// TwinCAT 3 PLC project MachineA
// ProgramVersion: 3.1.4026.22
// CompilerDefines: VISU_USEPROPERTYINFO
// libraries:
//   [DeviceLibrary], * (MechDS)
//   Tc2_MC2, * (Beckhoff Automation GmbH)
//   Tc2_Standard, * (Beckhoff Automation GmbH)
//   Tc2_System, * (Beckhoff Automation GmbH)
//   TcLog, * (Benedikt Geisler)
//   VisuSymbols, 4.5.0.0 (System)
// project tree:
//   / GlobalTextList.TcGTLO, PlcTask.TcTTO, Visualization Manager.TcVMO (not stored)
//   POUs/EquipmentModule1/ E_EquipmentModule1State.TcDUT, FB_EquipmentModule1.TcPOU, ST_EquipmentModuleFaults.TcDUT
//   POUs/EquipmentModule2/ E_EquipmentModule2State.TcDUT (not stored), FB_EquipmentModule2.TcPOU (not stored)
//   POUs/Machine/ E_ProductionState.TcDUT (not stored), FB_Machine.TcPOU (not stored)
//   POUs/ MAIN.TcPOU (not stored)
//   VISUs/ FB_Visu.TcPOU (not stored), PneumaticCylinder.TcVIS, Visualization.TcVIS
// real-time tasks:
//   TASK PlcTask: cycle T#10ms, priority 20, ADS port 350
//   TASK PlcTask1: cycle T#10ms, priority 21, ADS port 351
// motion (NC):
//   TASK NC-Task 1 SAF: cycle T#2ms, priority 4, ADS port 501
//   TASK NC-Task 1 SVB: cycle T#10ms, priority 8, ADS port 511
//   AXIS MachineAxis 1 (id 1)
//     OtherSettings: AllowMotionCmdToSlave=true
//     encoder EncType=16
//       EncPara: MaxCount=#x0000ffff
//     drive DrvType=13
//       Analog: TorqueSetpointScale=10, ScaleFactorActTorque=0.1
//       TimeComp: TaskDelayCycles=1
//     controller CtrType=1
//       CtrPara: PriorControlFactor=1
//         Observer: BandWidth=20
// variable links:
//   MachineA/MachineA Instance <-> NC-Task 1 SAF/Axes/MachineAxis 1
//     PlcTask Inputs/MAIN.fbMachine.fbEquipmentModule1.fbAxis1._axis.NcToPlc <-> Outputs/ToPlc
//     PlcTask Outputs/MAIN.fbMachine.fbEquipmentModule1.fbAxis1._axis.PlcToNc <-> Inputs/FromPlc
//   MachineA/MachineA Instance <-> MachineA_Sim/MachineA_Sim Instance
//     PlcTask Inputs/MAIN.fbMachine.fbEquipmentModule1.DoubleActingCylinderExtendSensor.HardwareInput <-> PlcTask Outputs/MAIN_SIM.bExtendSensor
//     PlcTask Inputs/MAIN.fbMachine.fbEquipmentModule1.DoubleActingCylinderRetractSensor.HardwareInput <-> PlcTask Outputs/MAIN_SIM.bRetractSensor
//     PlcTask Inputs/MAIN.fbMachine.fbEquipmentModule1.SingleActingCylinderExtendSensor.HardwareInput <-> PlcTask Outputs/MAIN_SIM.bExtendSensorSingle
//     PlcTask Inputs/MAIN.fbMachine.fbEquipmentModule1.SingleActingCylinderRetractSensor.HardwareInput <-> PlcTask Outputs/MAIN_SIM.bRetractSensorSingle
//     PlcTask Outputs/MAIN.fbMachine.fbEquipmentModule1.DoubleActingCylinderExtendSolenoid.HardwareOutput <-> PlcTask Inputs/MAIN_SIM.bExtendSolenoid
//     PlcTask Outputs/MAIN.fbMachine.fbEquipmentModule1.DoubleActingCylinderRetractSolenoid.HardwareOutput <-> PlcTask Inputs/MAIN_SIM.bRetractSolenoid
//     PlcTask Outputs/MAIN.fbMachine.fbEquipmentModule1.SingleActingCylinderExtendSolenoid.HardwareOutput <-> PlcTask Inputs/MAIN_SIM.bExtendSolenoidSingle

CONFIGURATION MachineA
    RESOURCE PLC ON TwinCAT3
        TASK PlcTask(INTERVAL := T#10ms, PRIORITY := 20);
        PROGRAM MAIN WITH PlcTask : MAIN;
    END_RESOURCE
END_CONFIGURATION

// ---- POUs/EquipmentModule1/E_EquipmentModule1State.TcDUT
{attribute 'qualified_only'}
{attribute 'strict'}
{attribute 'to_string'}
TYPE E_EquipmentModule1State :
(
    EXTEND_CYL1,
    WAIT_CYL1,
    EXTEND_CYL2,
    WAIT_CYL2,
    RETRACT_ALL,
    COMPLETE
);
END_TYPE

// ---- POUs/EquipmentModule1/ST_EquipmentModuleFaults.TcDUT
TYPE ST_EquipmentModuleFaults :
STRUCT
	ipEquipmentFault1 : I_Fault;
END_STRUCT
END_TYPE

// ---- POUs/EquipmentModule1/FB_EquipmentModule1.TcPOU
FUNCTION_BLOCK FB_EquipmentModule1 EXTENDS FB_MachineState IMPLEMENTS I_FaultOwner
VAR
    _subState : E_EquipmentModule1State;
	
	// Cylinder 1
    DoubleActingCylinderExtendSensor : FB_DigitalInputHardware(DebounceOnTime := T#0MS, DebounceOffTime := T#0MS, Invert := FALSE);
    DoubleActingCylinderRetractSensor : FB_DigitalInputHardware(DebounceOnTime := T#0MS, DebounceOffTime := T#0MS, Invert := FALSE);
    DoubleActingCylinderExtendSolenoid : FB_DigitalOutputHardware;
    DoubleActingCylinderRetractSolenoid : FB_DigitalOutputHardware;

    CylinderDoubleActing : FB_DoubleActingCylinder
	(
		iCylExtendedSwitch := DoubleActingCylinderExtendSensor,
		iCylRetractedSwitch := DoubleActingCylinderRetractSensor,
		iCylExtend := DoubleActingCylinderExtendSolenoid,
		iCylRetract := DoubleActingCylinderRetractSolenoid,
		eSensorMode := E_SensorMode.BOTH,
		tExtendTimeout := T#3S,
		tRetractTimeout := T#3S
	);

	// Cylinder 2
	_CylinderSingleActingIsInterlocked : BOOL; // Needed because you cant pass a Method as an interface
		
    SingleActingCylinderExtendSensor : FB_DigitalInputHardware(DebounceOnTime := T#0MS, DebounceOffTime := T#0MS, Invert := FALSE);
    SingleActingCylinderRetractSensor : FB_DigitalInputHardware(DebounceOnTime := T#0MS, DebounceOffTime := T#0MS, Invert := FALSE);
    SingleActingCylinderExtendSolenoid : FB_DigitalOutputHardware;

    CylinderSingleActing : FB_SingleActingCylinder
	(
		iCylExtendedSwitch := SingleActingCylinderExtendSensor,
		iCylRetractedSwitch := SingleActingCylinderRetractSensor,
		iCylExtend := SingleActingCylinderExtendSolenoid,
		eSensorMode := E_SensorMode.BOTH,
		tExtendTimeout := T#3S,
		tRetractTimeout := T#3S
	);
	
	// Cylinder Interfaces (not necessarily needed but makes changes easier) 
    iCylinder : I_Cylinder := CylinderDoubleActing; // Polymorphic reference				
    iCylinder2 : I_Cylinder := CylinderSingleActing; // Polymorphic reference

	// Axes
    fbAxis1 : FB_Axis;
	fbAxis2 : FB_Axis;

	// Faults
    fbFaultCyl1Extend : FB_Fault := (
        bAutoReset := FALSE,
        eSeverity := E_FaultSeverity.CRITICAL,
        nCode := 1001,
        sMessage := 'Cylinder 1 extend timeout'
    );
    fbFaultCyl1Retract : FB_Fault := (
        bAutoReset := FALSE,
        eSeverity := E_FaultSeverity.CRITICAL,
        nCode := 1002,
        sMessage := 'Cylinder 1 retract timeout'
    );
	fbFaultCyl1SensorConflict : FB_Fault := (
        bAutoReset := FALSE,
        eSeverity := E_FaultSeverity.CRITICAL,
        nCode := 1003,
        sMessage := 'Cylinder 1 sensor conflict'
    );
	
    fbFaultCyl2Extend  : FB_Fault := (
        bAutoReset := FALSE,
        eSeverity := E_FaultSeverity.CRITICAL,
        nCode := 1011,
        sMessage := 'Cylinder 2 extend timeout'
    );
    fbFaultCyl2Retract : FB_Fault := (
        bAutoReset := FALSE,
        eSeverity := E_FaultSeverity.CRITICAL,
        nCode := 1012,
        sMessage := 'Cylinder 2 retract timeout'
    );
    fbFaultCyl2SensorConflict : FB_Fault := (
        bAutoReset := FALSE,
        eSeverity := E_FaultSeverity.CRITICAL,
        nCode := 1013,
        sMessage := 'Cylinder 2 sensor conflict'
    );
	
	// Equiplevel Faults
    fbFaultSequenceTimeout : FB_Fault := (
        bAutoReset := FALSE,
        eSeverity := E_FaultSeverity.CRITICAL,
        nCode := 9999,
        sMessage := 'Equipment Module 1 Sequence Timeout'
    );
	
	_ipModuleFaults  : ST_EquipmentModuleFaults;
	
	fbFaultManager : FB_FaultManager;
END_VAR

PROPERTY AxisConveryor : I_Axis
GET
AxisConveryor := fbAxis1;
END_GET
END_PROPERTY

PROPERTY CylDouble : I_Cylinder
GET
CylDouble := CylinderDoubleActing;
END_GET
END_PROPERTY

PROPERTY CylSingle : I_Cylinder
GET
CylSingle := CylinderSingleActing;
END_GET
END_PROPERTY

METHOD ExecuteProduction
CASE _subState OF
    E_EquipmentModule1State.EXTEND_CYL1:
        _state := E_MachineState.RUNNING;  // transition from STARTING to RUNNING
        iCylinder.Extend();
        fbAxis1.MoveAbsolute(fPosition := 100.0, fVelocity := 50.0, fAccel := 10000.0, fDecel := 10000.0);
        _subState := E_EquipmentModule1State.WAIT_CYL1;

    E_EquipmentModule1State.WAIT_CYL1:
        IF iCylinder.IsExtended AND fbAxis1.IsIdle THEN
            _subState := E_EquipmentModule1State.EXTEND_CYL2;
        END_IF

    E_EquipmentModule1State.EXTEND_CYL2:
        iCylinder2.Extend();
        fbAxis1.MoveRelative(fDistance := -100.0, fVelocity := 500.0, fAccel := 1000.0, fDecel := 1000.0);
        _subState := E_EquipmentModule1State.WAIT_CYL2;

    E_EquipmentModule1State.WAIT_CYL2:
        IF iCylinder2.IsExtended AND fbAxis1.IsIdle THEN
            _subState := E_EquipmentModule1State.RETRACT_ALL;
        END_IF

    E_EquipmentModule1State.RETRACT_ALL:
        iCylinder.Retract();
        iCylinder2.Retract();
        IF iCylinder.IsRetracted AND iCylinder2.IsRetracted THEN
            _subState := E_EquipmentModule1State.COMPLETE;
        END_IF

    E_EquipmentModule1State.COMPLETE:
        _subState := E_EquipmentModule1State.EXTEND_CYL1;
        _state    := E_MachineState.IDLE;  // sequence done — back to IDLE
END_CASE
END_METHOD

METHOD ExecuteStop : BOOL
VAR_INPUT
END_VAR
// Command cylinders to retract
//iCylinder.Retract();
//iCylinder2.Retract();

// Hold axis
fbAxis1.Halt();

// Wait for everything to reach safe state
(*
IF iCylinder.IsRetracted AND iCylinder2.IsRetracted AND fbAxis.IsIdle THEN
	_subState := E_Module1State.EXTEND_CYL1;  // reset sequence
	_state    := E_MachineState.IDLE;
END_IF
*)
END_METHOD

PROPERTY FaultManager : POINTER TO FB_FaultManager
GET
FaultManager := ADR(fbFaultManager);
END_GET
END_PROPERTY

//FB_Init is always available implicitly and it is used primarily for initialization.
//The return value is not evaluated. For a specific influence, you can also declare the
//methods explicitly and provide additional code there with the standard initialization
//code. You can evaluate the return value.
METHOD FB_Init: BOOL
VAR_INPUT
    bInitRetains: BOOL; // TRUE: the retain variables are initialized (reset warm / reset cold)
    bInCopyCode: BOOL;  // TRUE: the instance will be copied to the copy code afterward (online change)   
END_VAR
VAR
	stFaults : ST_CylinderFaults;
END_VAR
CylinderSingleActing.SetInterlock(_CylinderSingleActingIsInterlocked);

// Inject faults into cylinders
stFaults.ipFaultExtend := fbFaultCyl1Extend;
stFaults.ipFaultRetract := fbFaultCyl1Retract;
stFaults.ipFaultSensorConflict := fbFaultCyl1SensorConflict;
CylinderDoubleActing.SetFaults(stFaults);

stFaults.ipFaultExtend  := fbFaultCyl2Extend;
stFaults.ipFaultRetract := fbFaultCyl2Retract;
stFaults.ipFaultSensorConflict := 0;
CylinderSingleActing.SetFaults(stFaults);

fbFaultManager.RegisterFault(fbFaultCyl1Extend);
fbFaultManager.RegisterFault(fbFaultCyl1Retract);
fbFaultManager.RegisterFault(fbFaultCyl1SensorConflict);
fbFaultManager.RegisterFault(fbFaultCyl2Extend);
fbFaultManager.RegisterFault(fbFaultCyl2Retract);
fbFaultManager.RegisterFault(fbFaultCyl2SensorConflict);
END_METHOD

METHOD RegisterFaults
VAR_INPUT
	ipManager : I_FaultManager;
END_VAR
ipManager.RegisterFault(fbFaultSequenceTimeout);
END_METHOD

METHOD Reset : BOOL
CylDouble.Reset();
CylSingle.Reset();
AxisConveryor.Reset();
END_METHOD

METHOD Run
// Raise Equipment Level Faults
IF _ipModuleFaults.ipEquipmentFault1 <> 0 THEN
	_ipModuleFaults.ipEquipmentFault1.Raise();
END_IF

iCylinder.Run();
iCylinder2.Run();
fbAxis1.Run();
fbAxis2.Run();

_CylinderSingleActingIsInterlocked := iCylinder.IsRetracted;

// Check faults
fbFaultManager.Run();

CASE _state OF
	E_MachineState.IDLE:
		;
	E_MachineState.RUNNING:
		THIS^.ExecuteProduction();
	E_MachineState.STOPPING:
		THIS^.ExecuteStop();
END_CASE
END_METHOD

END_FUNCTION_BLOCK

// ---- GlobalTextList.TcGTLO
TEXTLIST GlobalTextList
  717 = 'Cylinders'
  189 = 'Enable'
  830 = 'Enable Axis'
  77 = 'Ext'
  96 = "Ext'd"
  384 = 'Extend'
  59 = 'Extend Cylinder'
  82 = 'Extended'
  464 = 'Fault'
  635 = 'Feedback'
  309 = 'Feedbacks'
  997 = 'Home'
  144 = 'Home Axis'
  673 = 'Motor Axis'
  684 = 'Reset'
  101 = "Ret'd"
  630 = 'Retract'
  87 = 'Retracted'
  116 = 'Run'
  703 = 'Run Sequence'
  870 = 'Solenoid'
  744 = 'Solenoids'
END_TEXTLIST

// ---- VISUs/PneumaticCylinder.TcVIS
VISUALIZATION PneumaticCylinder  // 1024x768
END_VISUALIZATION

// ---- VISUs/Visualization.TcVIS
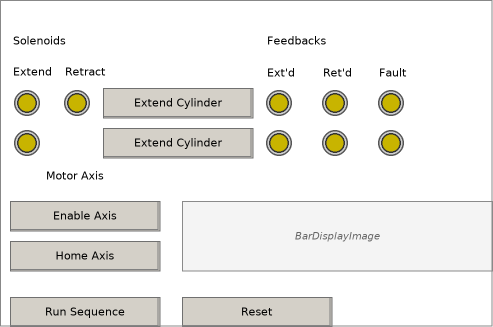
VISUALIZATION Visualization  // 493x327
    Button (103,88 150x30), "Extend Cylinder"
        toggle MAIN.fbVisu.bButtonExtendDouble
    Lamp1 (62,88 30x30), variable: MAIN.fbMachine.fbEquipmentModule1.CylinderDoubleActing._cmdRetract, style: Lamp-Lamp1-Yellow
    Lamp1 (12,88 30x30), variable: MAIN.fbMachine.fbEquipmentModule1.CylinderDoubleActing._cmdExtend, style: Lamp-Lamp1-Yellow
    Lamp1 (320,88 30x30), variable: (MAIN.fbMachine.fbEquipmentModule1.CylinderDoubleActing._state=E_CylinderState.RETRACTED), style: Lamp-Lamp1-Yellow
    Lamp1 (264,88 30x30), variable: (MAIN.fbMachine.fbEquipmentModule1.CylinderDoubleActing._state=E_CylinderState.EXTENDED), style: Lamp-Lamp1-Yellow
    Button (103,128 150x30), "Extend Cylinder"
        toggle MAIN.fbVisu.bButtonExtendSingle
    Lamp1 (12,128 30x30), variable: MAIN.fbMachine.fbEquipmentModule1.CylinderSingleActing._cmdExtend, style: Lamp-Lamp1-Yellow
    Lamp1 (320,128 30x30), variable: (MAIN.fbMachine.fbEquipmentModule1.CylinderSingleActing._state=E_CylinderState.RETRACTED), style: Lamp-Lamp1-Yellow
    Lamp1 (264,128 30x30), variable: (MAIN.fbMachine.fbEquipmentModule1.CylinderSingleActing._state=E_CylinderState.EXTENDED), style: Lamp-Lamp1-Yellow
    Button (10,297 150x30), "Run Sequence"
        toggle MAIN.fbVisu.bButtonRunProduction
    Button (182,297 150x30), "Reset"
        toggle MAIN.fbVisu.bButtonReset
    BarDisplayImage (182,201 311x70), value: MAIN.fbMachine.fbEquipmentModule1.fbAxis1._axis.NcToPlc.ActPos, style: BarDisplayImage-Gray, scale format: %.1f, scale 0..100
    Button (10,201 150x30), "Enable Axis"
        toggle MAIN.fbVisu.bButtonEnableAxis
    Button (10,241 150x30), "Home Axis"
        toggle MAIN.fbVisu.bButtonHomeAxis
    Label (264,26 70x30), "Feedbacks"
    Label (10,26 70x30), "Solenoids"
    Label (0,161 150x30), "Motor Axis"
    Label (10,57 45x30), "Extend"
    Label (62,57 55x30), "Retract"
    Label (320,58 62x30), "Ret'd"
    Label (264,58 64x30), "Ext'd"
    Lamp1 (376,88 30x30), variable: MAIN.fbMachine.fbEquipmentModule1.CylinderDoubleActing._isFaulted, style: Lamp-Lamp1-Yellow
    Label (376,58 62x30), "Fault"
    Lamp1 (376,128 30x30), variable: MAIN.fbMachine.fbEquipmentModule1.CylinderSingleActing._isFaulted, style: Lamp-Lamp1-Yellow
END_VISUALIZATION
